(* PLC project Generated.project, CODESYS CODESYS V3.5 SP19 Patch 1 *)
(* stored: creationDateTime 2026-08-11T18:19:14.781842, modificationDateTime 2026-08-11T18:19:14.781842 *)

(* ═══════════════════════════════════════════════════════════════ 🏗️ ST_HardwareImage — Structure globale d'image matérielle (Frontière HwIn) ─────────────────────────────────────────────────────────────── 📄 Lot L5 (Frontière unique HwIn) 🎨 Agrège les 4 sous-domaines matériels : Winch, Translation, Operator, Machine. ═══════════════════════════════════════════════════════════════ *)
TYPE ST_HardwareImage : STRUCT
  Winch : ST_HwWinch;  (* Entrées brutes domaine Treuils M1/M2 + codeurs *)
  Translation : ST_HwTranslation;  (* Entrées brutes domaine Translation M3 + variateur *)
  Operator : ST_HwOperator;  (* Entrées brutes domaine Opérateur / Joystick / bus CAN *)
  Machine : ST_HwMachine;  (* Entrées brutes domaine Sécurités/Communs Machine *)
END_STRUCT;
END_TYPE

(* ═══════════════════════════════════════════════════════════════ 🏗️ ST_HwMachine — Image matérielle brute des entrées communes Machine ─────────────────────────────────────────────────────────────── 📄 Lot L5 (Frontière unique HwIn) 🎨 Regroupe les signaux physiques d'entrée bruts communs à la machine. ═══════════════════════════════════════════════════════════════ *)
TYPE ST_HwMachine : STRUCT
  PowerContactorEngaged_DI : BOOL;  (* Confirm. contacteur puissance engagé *)
  EmergencyChainClosed_DI : BOOL;  (* Boucle AU fermée (coup-de-poing + contact PLC) *)
  PhaseRotationOk_DI : BOOL;  (* Contrôle rotation phases élec. OK *)
  BrakeThermalOk_DI : BOOL;  (* Thermique frein M1/M2/M3 commun OK *)
  M1_M2_KoboldContactFond_DI : BOOL;  (* Retour détecteur fond Kobold *)
  HydraulicThermalOk_DI : BOOL;  (* Thermique centrale hydraulique OK *)
  ConveyorInfeedReady_DI : BOOL;  (* Autorisation démarrage crible (dépôt gravats) *)
END_STRUCT;
END_TYPE

(* ═══════════════════════════════════════════════════════════════ 🏗️ ST_HwOperator — Image matérielle brute des entrées Opérateur / Joystick ─────────────────────────────────────────────────────────────── 📄 Lot L5 (Frontière unique HwIn) 🎨 Regroupe les signaux physiques d'entrée bruts du joystick CANopen JOY1. ═══════════════════════════════════════════════════════════════ *)
TYPE ST_HwOperator : STRUCT
  JoyXRaw_ANA1 : INT;  (* Valeur brute analogique axe X (Translation) *)
  JoyYRaw_ANA2 : INT;  (* Valeur brute analogique axe Y (Levage) *)
  JoyBtnRaw : BOOL;  (* Bouton brut joystick (Homme-Mort) *)
  CanBusState : INT;  (* État bus CANopen (CANbus.GetBusState) *)
  JOY1_DeviceState : DEVICE_STATE;  (* État device JOY1 (GetDeviceState) *)
END_STRUCT;
END_TYPE

(* ═══════════════════════════════════════════════════════════════ 🏗️ ST_HwTranslation — Image matérielle brute des entrées Translation M3 ─────────────────────────────────────────────────────────────── 📄 Lot L5 (Frontière unique HwIn) 🎨 Regroupe les signaux physiques d'entrée bruts de la translation M3 (AC600). ═══════════════════════════════════════════════════════════════ *)
TYPE ST_HwTranslation : STRUCT
  M3_PosTremie_DI : BOOL;  (* Capteur position trémie *)
  M3_PosPV_DI : BOOL;  (* Capteur position point de vitesse (pré-ralentissement) *)
  M3_PosP2_DI : BOOL;  (* Capteur position P2 *)
  M3_PosP1_DI : BOOL;  (* Capteur position P1 *)
  M3_PosMaintenance_DI : BOOL;  (* Capteur position maintenance *)
  M3_BrakeIsOpen_DI : BOOL;  (* Retour frein M3 (1 = ouvert) *)
  M3_ThermalOK_DI : BOOL;  (* 🆕 T96 : retour disjoncteur thermique moteur/variateur AC600 (1 = OK, même polarité que BrakeThermalFeedback/M1/M2ThermalFeedback) — diagnostic seul, l'AC600 se protège déjà lui-même *)
  M3_StatusWord : WORD;  (* Status word variateur AC600 *)
  M3_ActualFrequencyHz : UINT;  (* Fréquence réelle variateur AC600 (x100) *)
  AC600_DeviceState : DEVICE_STATE;  (* État device AC600 (GetDeviceState) *)
END_STRUCT;
END_TYPE

(* ═══════════════════════════════════════════════════════════════ 🏗️ ST_HwWinch — Image matérielle brute des entrées Treuils M1 / M2 ─────────────────────────────────────────────────────────────── 📄 Lot L5 (Frontière unique HwIn) 🎨 Regroupe les signaux physiques d'entrée bruts des treuils M1 et M2. ═══════════════════════════════════════════════════════════════ *)
TYPE ST_HwWinch : STRUCT
  M1_ContactorsReleased_DI : BOOL;  (* Retours contacteurs M1 retombés *)
  M1_ThermalOk_DI : BOOL;  (* Thermique moteur M1 OK *)
  M1_BrakeIsOpen_DI : BOOL;  (* Retour frein M1 (1 = ouvert) *)
  M2_ContactorsReleased_DI : BOOL;  (* Retours contacteurs M2 retombés *)
  M2_ThermalOk_DI : BOOL;  (* Thermique moteur M2 OK *)
  M2_BrakeIsOpen_DI : BOOL;  (* Retour frein M2 (1 = ouvert) *)
  M1M2_TopPositionFree_DI : BOOL;  (* Capteur position haute commun M1/M2 libre *)
  M2_TensionedCable_DI : BOOL;  (* Capteur mou de câble M2 (câble tendu) *)
  COD1_PosValue : UDINT;  (* Valeur brute position codeur COD1 (M1) *)
  COD1_Alarms : UINT;  (* Alarmes brutes COD1 *)
  COD1_Warnings : UINT;  (* Avertissements bruts COD1 *)
  COD1_DeviceState : DEVICE_STATE;  (* État device COD1 (GetDeviceState) *)
  COD2_PosValue : UDINT;  (* Valeur brute position codeur COD2 (M2) *)
  COD2_Alarms : UINT;  (* Alarmes brutes COD2 *)
  COD2_Warnings : UINT;  (* Avertissements bruts COD2 *)
  COD2_DeviceState : DEVICE_STATE;  (* État device COD2 (GetDeviceState) *)
END_STRUCT;
END_TYPE

(* ═══════════════════════════════════════════════════════════════ 🧪 FB_SimBench — Enveloppe unique de simulation pour banc d'essai ─────────────────────────────────────────────────────────────── 📄 Doc métier : DOC/AF/AF_Partie-13_Fonction_Simulation_v2.1.md 📄 Lot L6 (Rebranchement du banc de simulation derrière HwIn) 🎯 Rôle : Compose les 4 blocs de modèle de simulation existants : - FB_Sim_Encoder (instM1, instM2) - FB_Sim_Translation (instTranslation) - FB_Sim_Joystick (instJoystick) - FB_Sim_Safety (instSafety) 🔒 Brique réduite : 0 lecture de variable globale en interne. Toutes les entrées (commandes, stimuli, HwReal) sont passées en paramètres. 🔴 RÈGLES SÉCURITÉ ET POLARITÉ : - Modèle frein M1/M2/M3 : M1_BrakeIsOpen_DI := M1_BrakeCmd (1 = OUVERT). Ne JAMAIS faire NOT BrakeCmd ! (P1 Lot L6). - Retours contacteurs M1/M2 : 1 = tous retombés (TRUE quand RelayFwd=0 et RelayRev=0). ═══════════════════════════════════════════════════════════════ *)
FUNCTION_BLOCK FB_SimBench
  VAR_INPUT
    Enable : BOOL;  (* Activation globale (GVL_Simulation.SimulationModeActive) *)
    M1_RelayFwd : BOOL;  (* ── Commandes issues de l'automate (Scan N-1 / PRG_07 / PRG_10) ────────── *)
    M1_RelayRev : BOOL;
    M1_SpeedContactor_1 : BOOL;  (* 🔧 REX 2026-07-27 : les 4 contacteurs de palier participent au retour unique « tous contacteurs retombés » — sans eux, le modèle annonce l'arrêt alors qu'un palier est encore engagé (fausse condition d'armement Méca A). *)
    M1_SpeedContactor_2 : BOOL;
    M1_SpeedContactor_3 : BOOL;
    M1_SpeedContactor_4 : BOOL;
    M1_SpeedRefPct : REAL;
    M1_PresetTriggerCmd : WORD;
    M1_PresetValueOut : UDINT;
    M1_BrakeCmd : BOOL;  (* TRUE = commande desserrage frein M1 *)
    M2_RelayFwd : BOOL;
    M2_RelayRev : BOOL;
    M2_SpeedContactor_1 : BOOL;  (* 🔧 REX 2026-07-27 : idem M1, voir ci-dessus *)
    M2_SpeedContactor_2 : BOOL;
    M2_SpeedContactor_3 : BOOL;
    M2_SpeedContactor_4 : BOOL;
    M2_SpeedRefPct : REAL;
    M2_PresetTriggerCmd : WORD;
    M2_PresetValueOut : UDINT;
    M2_BrakeCmd : BOOL;  (* TRUE = commande desserrage frein M2 *)
    M3_Direction : INT;  (* 1 = Avant, -1 = Arrière, 0 = Arrêt *)
    M3_SpeedRefPct : REAL;
    M3_BrakeCmd : BOOL;  (* TRUE = commande desserrage frein M3 *)
    M3_TargetNum : INT;  (* Cible sélectionnée (0..4) *)
    PowerKeepAlive_A : BOOL;  (* TRUE = relais A maintenu sagement par le PLC *)
    PowerKeepAlive_B : BOOL;  (* TRUE = relais B maintenu sagement par le PLC *)
    EmergencyArming_RQ : BOOL;  (* Impulsion de réarmement puissance *)
    SimEncoderSpeedFactor : REAL := 1;  (* ── Stimuli & Paramètres de banc ───────────────────────────────────────── *)
    SimSyncDeviationInjectM1 : BOOL := FALSE;
    SimSyncDeviationInjectM2 : BOOL := FALSE;
    SimSyncDeviationOffset_M : REAL := 0.5;
    SimM3SensorsWordActive : BOOL := FALSE;
    SimM3SensorsWord : BYTE := 16#01;
    SimJoystickRawX : INT := 5000;
    SimJoystickRawY : INT := 5000;
    SimJoystickRawButton : BOOL := FALSE;
    SimKoboldContactValue : BOOL := FALSE;
    BtnEmergencyStop : BOOL := FALSE;  (* Simulation appui coup-de-poing AU *)
    HwReal : ST_HardwareImage;  (* ── Image réelle fallback ──────────────────────────────────────────────── *)
  END_VAR
  VAR_OUTPUT
    Winch : ST_HwWinch;
    Translation : ST_HwTranslation;
    Operator : ST_HwOperator;
    Machine : ST_HwMachine;
  END_VAR
  VAR_IN_OUT
    RawPosM1 : UDINT;  (* Mémoire _SimEncoderRawPosM1 dans GVL_PERSISTENT *)
    RawPosM2 : UDINT;  (* Mémoire _SimEncoderRawPosM2 dans GVL_PERSISTENT *)
  END_VAR
  VAR
    instSimEncoderM1 : FB_Sim_Encoder;  (* Modèles sous-jacents *)
    instSimEncoderM2 : FB_Sim_Encoder;
    instSimTranslation : FB_Sim_Translation;
    instSimJoystick : FB_Sim_Joystick;
    instSimSafety : FB_Sim_Safety;
    M1_PresetCmd : BOOL;  (* Calculs internes *)
    M2_PresetCmd : BOOL;
    M1_OffsetPts : DINT;
    M2_OffsetPts : DINT;
    M3_RelayFwd : BOOL;
    M3_RelayRev : BOOL;
    M3_ActualFreqHz : UINT;
    M3_StatusWordSim : WORD;
  END_VAR

            

// === IMPLEMENTATION ===

IF NOT Enable THEN
    Winch       := HwReal.Winch;
    Translation := HwReal.Translation;
    Operator    := HwReal.Operator;
    Machine     := HwReal.Machine;
    RETURN;
END_IF;


// ── 1. MODÈLE TREUILS (M1 + M2) ─────────────────────────────────────────────
// Presets codeurs : déclenchés si PresetTriggerCmd = 2
M1_PresetCmd := (M1_PresetTriggerCmd = 2);
M2_PresetCmd := (M2_PresetTriggerCmd = 2);

// Conversions d'injection d'écart synchro (0.5m -> points codeur avec 8192 pts/tour, 2m/tour)
// 1m = 4096 points codeur.
M1_OffsetPts := REAL_TO_DINT(SimSyncDeviationOffset_M * 4096.0);
M2_OffsetPts := REAL_TO_DINT(SimSyncDeviationOffset_M * 4096.0);

// Instance modèle codeur M1
instSimEncoderM1(
    Enable           := TRUE,
    RelayFwd         := M1_RelayFwd,
    RelayRev         := M1_RelayRev,
    SpeedRefPct      := M1_SpeedRefPct,
    PresetCmd        := M1_PresetCmd,
    PresetValue      := M1_PresetValueOut,
    SpeedScaleFactor := SimEncoderSpeedFactor,
    TestOffsetCmd    := SimSyncDeviationInjectM1,
    TestOffsetPts    := M1_OffsetPts,
    RawPos           := RawPosM1
);

// Instance modèle codeur M2
instSimEncoderM2(
    Enable           := TRUE,
    RelayFwd         := M2_RelayFwd,
    RelayRev         := M2_RelayRev,
    SpeedRefPct      := M2_SpeedRefPct,
    PresetCmd        := M2_PresetCmd,
    PresetValue      := M2_PresetValueOut,
    SpeedScaleFactor := SimEncoderSpeedFactor,
    TestOffsetCmd    := SimSyncDeviationInjectM2,
    TestOffsetPts    := M2_OffsetPts,
    RawPos           := RawPosM2
);

// Recopie structures Winch simulées :
// 🛑 POLARITÉ DE FREIN SIMULÉ (P1 Lot L6) : 1 = contacteur commandé = frein OUVERT.
// Câblage réel : DI = 1 ⟺ frein OUVERT. Le modèle produit donc M1_BrakeIsOpen_DI := M1_BrakeCmd !
Winch.M1_BrakeIsOpen_DI        := M1_BrakeCmd;
// 🔧 REX 2026-07-27 : retour UNIQUE « tous contacteurs retombés » = sens ET vitesse.
// Omettre les paliers ferait croire à l'arrêt pendant les transitoires → Méca A armée à tort.
Winch.M1_ContactorsReleased_DI := NOT (M1_RelayFwd OR M1_RelayRev
                                    OR M1_SpeedContactor_1 OR M1_SpeedContactor_2
                                    OR M1_SpeedContactor_3 OR M1_SpeedContactor_4);
Winch.M1_ThermalOk_DI          := TRUE; // Sauf panne simulée

Winch.M2_BrakeIsOpen_DI        := M2_BrakeCmd;
Winch.M2_ContactorsReleased_DI := NOT (M2_RelayFwd OR M2_RelayRev
                                    OR M2_SpeedContactor_1 OR M2_SpeedContactor_2
                                    OR M2_SpeedContactor_3 OR M2_SpeedContactor_4);
Winch.M2_ThermalOk_DI          := TRUE;

Winch.M1M2_TopPositionFree_DI  := TRUE; // Butée libre au repos en simu
Winch.M2_TensionedCable_DI     := TRUE; // Câble tendu en simu

Winch.COD1_PosValue            := instSimEncoderM1.RawPosOut;
Winch.COD1_Alarms              := 0;
Winch.COD1_Warnings            := 0;
Winch.COD1_DeviceState         := 4; // DEVICE_STATE RUNNING = 4 (bus OK)

Winch.COD2_PosValue            := instSimEncoderM2.RawPosOut;
Winch.COD2_Alarms              := 0;
Winch.COD2_Warnings            := 0;
Winch.COD2_DeviceState         := 4; // DEVICE_STATE RUNNING = 4


// ── 2. MODÈLE TRANSLATION M3 (AC600) ─────────────────────────────────────────
M3_RelayFwd := (M3_Direction = 1);
M3_RelayRev := (M3_Direction = -1);

instSimTranslation(
    Enable      := TRUE,
    TargetNum   := M3_TargetNum,
    RelayFwd    := M3_RelayFwd,
    RelayRev    := M3_RelayRev,
    TravelTimeS := 8.0,
    PVLeadTimeS := 2.0
);

// Remplissage capteurs de position M3 :
IF SimM3SensorsWordActive THEN
    Translation.M3_PosTremie_DI      := SimM3SensorsWord.0;
    Translation.M3_PosPV_DI          := SimM3SensorsWord.1;
    Translation.M3_PosP2_DI          := SimM3SensorsWord.2;
    Translation.M3_PosP1_DI          := SimM3SensorsWord.3;
    Translation.M3_PosMaintenance_DI := SimM3SensorsWord.4;
ELSE
    Translation.M3_PosTremie_DI      := instSimTranslation.PosTremie;
    Translation.M3_PosPV_DI          := instSimTranslation.PosPV;
    Translation.M3_PosP2_DI          := instSimTranslation.PosP2;
    Translation.M3_PosP1_DI          := instSimTranslation.PosP1;
    Translation.M3_PosMaintenance_DI := instSimTranslation.PosMaintenance;
END_IF;

// Polarité frein M3 (1 = OUVERT)
Translation.M3_BrakeIsOpen_DI    := M3_BrakeCmd;

// 🆕 T96 : thermique moteur/variateur AC600 — pas de panne simulée, toujours OK (comme Winch.M1/M2_ThermalOk_DI)
Translation.M3_ThermalOK_DI      := TRUE;

// Simulation StatusWord AC600 : Bit 0 (Power Ready) = 1, Bit 7 (Comm Ready) = 1 -> 16#0081
IF (M3_Direction <> 0) THEN
    M3_StatusWordSim := 16#0087; // + Operating/Running
    M3_ActualFreqHz  := REAL_TO_UINT(M3_SpeedRefPct * 50.0); // 50.0 Hz à 100% (x100 -> 5000)
ELSE
    M3_StatusWordSim := 16#0081;
    M3_ActualFreqHz  := 0;
END_IF;

Translation.M3_StatusWord        := M3_StatusWordSim;
Translation.M3_ActualFrequencyHz := M3_ActualFreqHz;
Translation.AC600_DeviceState    := 4; // DEVICE_STATE RUNNING = 4


// ── 3. MODÈLE OPÉRATEUR / JOYSTICK ───────────────────────────────────────────
instSimJoystick(
    Enable     := TRUE,
    NeutralRaw := 5000,
    MaxRaw     := 10000
);

// Permet aux stimuli de banc de surcharger le retour du joystick si spécifié :
IF SimJoystickRawX <> 5000 THEN
    Operator.JoyXRaw_ANA1 := SimJoystickRawX;
ELSE
    Operator.JoyXRaw_ANA1 := instSimJoystick.RawX;
END_IF;

IF SimJoystickRawY <> 5000 THEN
    Operator.JoyYRaw_ANA2 := SimJoystickRawY;
ELSE
    Operator.JoyYRaw_ANA2 := instSimJoystick.RawY;
END_IF;

IF SimJoystickRawButton THEN
    Operator.JoyBtnRaw := TRUE;
ELSE
    Operator.JoyBtnRaw := instSimJoystick.RawButton;
END_IF;

Operator.CanBusState      := 2; // CANbusState 2 = ACTIVE (confirmé terrain)
Operator.JOY1_DeviceState := 4; // DEVICE_STATE RUNNING = 4


// ── 4. MODÈLE SÉCURITÉ & COMMUNS MACHINE ─────────────────────────────────────
instSimSafety(
    Enable           := TRUE,
    PowerCutOff_A    := PowerKeepAlive_A,
    PowerCutOff_B    := PowerKeepAlive_B,
    EmergencyArming  := EmergencyArming_RQ,
    BtnEmergencyStop := BtnEmergencyStop
);

Machine.PowerContactorEngaged_DI   := instSimSafety.SimContactorOk;
Machine.EmergencyChainClosed_DI    := instSimSafety.SimChainOk;
Machine.PhaseRotationOk_DI         := TRUE;
Machine.BrakeThermalOk_DI          := TRUE;
Machine.M1_M2_KoboldContactFond_DI := SimKoboldContactValue;
Machine.HydraulicThermalOk_DI      := TRUE;

          
END_FUNCTION_BLOCK

(* ═══════════════════════════════════════════════════════════════ 🧪 FB_Sim_Encoder — Simulation physique d'un codeur absolu de treuil ─────────────────────────────────────────────────────────────── 📄 Doc métier : DOC/AF/AF_Partie-13_Fonction_Simulation_v2.1.md 🧩 Brique réduite (Partie3 §1bis, "briques E/S & diagnostics") : pas de contrat Enable/Reset/Error complet, pas de StartStop/SafeStop — outil de banc, pas du métier machine. 🎯 Rôle : fait "compter" un codeur absolu comme si le treuil tournait réellement, à partir des relais de sens commandés et de la vitesse rampée courante. Extraction PURE de la logique déjà en place dans `PRG_02_Encoders.st` (bloc "SIMULATION SUR BANC DE TEST") — aucun changement de comportement, juste la dissociation en FB dédié. 📥 Enable : simulation active (SimulationModeActive AND NOT BusEncoderMxIsReal) 📥 RelayFwd/RelayRev : sens commandé (contacteurs de sens du treuil) 📥 SpeedRefPct : vitesse rampée courante (magnitude, %) — ex. instWinchM1.SpeedRamp.Current 📥 PresetCmd : TRUE le cycle où un preset (homing) doit être appliqué (PresettTrigCmd = 2) 📥 PresetValue : valeur brute à charger lors du preset 📥 SpeedScaleFactor : 🔧 REX 2026-07-07 — multiplicateur de vitesse simulation (confort de test banc uniquement, sans rapport avec une calibration réelle). Défaut 1.0 = comportement d'origine. Câblé sur GVL_Simulation.TstEncoderSpeedFactor (réglable à chaud, sans recompiler). 📤 RawPosOut : position brute simulée (UDINT), à aiguiller à la place de la valeur EtherCAT réelle quand le device n'est pas Operational (voir PRG_02_Encoders.st) 🔧 REX 2026-07-08 : `RawPos` déplacé en `VAR_IN_OUT`, référencé depuis `GVL_PERSISTENT` (même pattern que `Calib` dans `FB_Encoder_Homing`) — `PERSISTENT` n'est valide que sur du `VAR_GLOBAL` en CODESYS, pas sur une variable locale de FB (tenté en `VAR RETAIN` puis `VAR PERSISTENT RETAIN` locaux, aucun des deux ne convient). Un vrai codeur absolu physique conserve son comptage brut même à travers un reset FROID (indépendant de l'automate) — il fallait donc bien du PERSISTENT RETAIN réel, regroupé avec le reste dans GVL_PERSISTENT. ═══════════════════════════════════════════════════════════════ === DECLARATION (à coller dans la partie déclaration du POU FB_Sim_Encoder) === *)
FUNCTION_BLOCK FB_Sim_Encoder
  VAR_INPUT
    Enable : BOOL;
    RelayFwd : BOOL;
    RelayRev : BOOL;
    SpeedRefPct : REAL;
    PresetCmd : BOOL;
    PresetValue : UDINT;
    SpeedScaleFactor : REAL := 1;  (* 🔧 REX 2026-07-07 — confort de test, voir bandeau ci-dessus *)
    TestOffsetCmd : BOOL;  (* 🆕 REX 2026-07-08 (4) — front montant = applique TestOffsetPts (test banc) *)
    TestOffsetPts : DINT := 0;  (* 🆕 REX 2026-07-08 (4) — décalage signé à appliquer (points bruts) *)
  END_VAR
  VAR_OUTPUT
    RawPosOut : UDINT;
  END_VAR
  VAR_IN_OUT
    RawPos : UDINT;  (* 🔧 REX 2026-07-08 : référence _SimEncoderRawPosM1/M2 (survit au reset froid) *)
  END_VAR
  VAR
    Increment : UDINT;  (* 🔧 REX 2026-07-07 — évite de dupliquer le calcul 2x *)
    TestOffsetEdge : R_TRIG;  (* 🆕 REX 2026-07-08 (4) *)
  END_VAR

            

// === IMPLEMENTATION (à coller dans le corps ST du POU FB_Sim_Encoder) ===

IF NOT Enable THEN
    RawPosOut := RawPos;
    RETURN;
END_IF;

// 🆕 REX 2026-07-08 (4) — injection test banc : VRAI saut de position (comme un glissement réel),
// pour tester Concept 1 / Méca E ET le rattrapage joystick (voir GVL_Simulation bandeau).
TestOffsetEdge(CLK := TestOffsetCmd);
IF TestOffsetEdge.Q THEN
    RawPos := DINT_TO_UDINT(UDINT_TO_DINT(RawPos) + TestOffsetPts);
END_IF;

Increment := REAL_TO_UDINT(SpeedRefPct * 0.1 * SpeedScaleFactor);

IF PresetCmd THEN
    RawPos := PresetValue;
ELSIF RelayFwd THEN
    RawPos := RawPos + Increment;
ELSIF RelayRev THEN
    IF RawPos >= Increment THEN
        RawPos := RawPos - Increment;
    ELSE
        RawPos := 0;
    END_IF;
END_IF;

RawPosOut := RawPos;

          
END_FUNCTION_BLOCK

(* ═══════════════════════════════════════════════════════════════ 🧪 FB_Sim_Joystick — Simulation des entrées brutes joystick (bus CAN hors ligne) ─────────────────────────────────────────────────────────────── 📄 Doc métier : DOC/AF/AF_Partie-13_Fonction_Simulation_v2.1.md 🧩 Brique réduite (Partie3 §1bis) : outil de banc, pas du métier machine. 🎯 Rôle : remplace l'ancien bypass homme-mort codé en dur dans `FB_Joystick` (`GVL_DEBUG.DBG_DeadmanBypass_TEST`, qui forçait `DeadmanArmed` en permanence — un vrai contournement de sécurité). Ici, on simule les ENTRÉES BRUTES du capteur (`RawX`/`RawY`/`RawButton`) : le homme-mort réel de `FB_Joystick` reste pleinement actif et doit toujours être "actionné" (forcer `RawButton` en instance CODESYS) pour armer — comportement métier testé pour de vrai, pas contourné. 📥 Enable : simulation active (SimulationModeActive AND NOT BusJoystickSignalIsReal) — 🔧 REX 2026-07-08 : granularité séparée du bus CANopen (BusJoystickIsReal, voir GVL_Simulation) 📥 NeutralRaw : valeur brute simulée au repos (voir GVL_Simulation.TstJoystickForceNeutralRaw) 📥 MaxRaw : valeur brute simulée à fond (voir GVL_Simulation.TstJoystickForceMaxRaw) 📤 RawX/RawY : forçables en instance CODESYS (par défaut = NeutralRaw, repos) 📤 RawButton : forçable en instance CODESYS (par défaut = FALSE, relâché) 💡 Note d'application : en vue instance CODESYS, forcer `RawX`/`RawY` à `MaxRaw` (ou une valeur intermédiaire) pour simuler un débattement, et `RawButton` à `TRUE` pour simuler l'appui homme-mort — exactement comme on forcerait le vrai capteur. ═══════════════════════════════════════════════════════════════ === DECLARATION (à coller dans la partie déclaration du POU FB_Sim_Joystick) === *)
FUNCTION_BLOCK FB_Sim_Joystick
  VAR_INPUT
    Enable : BOOL;
    NeutralRaw : INT := 5000;
    MaxRaw : INT := 10000;
  END_VAR
  VAR_OUTPUT
    RawX : INT;  (* 🔧 Forçable en instance CODESYS (repos = NeutralRaw) *)
    RawY : INT;  (* 🔧 Forçable en instance CODESYS (repos = NeutralRaw) *)
    RawButton : BOOL;  (* 🔧 Forçable en instance CODESYS (repos = FALSE) *)
  END_VAR
  VAR
    FirstCycle : BOOL := TRUE;
  END_VAR

            

// === IMPLEMENTATION (à coller dans le corps ST du POU FB_Sim_Joystick) ===

// 🔑 Initialise au neutre au premier cycle uniquement — ensuite RawX/RawY/RawButton
// restent forçables librement en instance CODESYS (un Force n'est jamais écrasé par TRUE,
// mais une simple écriture cyclique l'écraserait — donc pas de ré-assignation continue ici).
IF NOT Enable THEN
    FirstCycle := TRUE;
    RETURN;
END_IF;

IF FirstCycle THEN
    RawX := NeutralRaw;
    RawY := NeutralRaw;
    RawButton := FALSE;
    FirstCycle := FALSE;
END_IF;

          
END_FUNCTION_BLOCK

(* ═══════════════════════════════════════════════════════════════ 🧪 FB_Sim_Safety — Simulation de la chaîne d'AU et du contacteur de puissance ─────────────────────────────────────────────────────────────── 📥 Enable : activation de la simulation (SimulationModeActive AND NOT SensorEmergencyStopChainIsReal) 📥 PowerCutOff_A : demande de coupure PLC canal A (maintenu à TRUE en marche normale) 📥 PowerCutOff_B : demande de coupure PLC canal B (maintenu à TRUE en marche normale) 📥 EmergencyArming : impulsion de réarmement (EmergencyArming_RQ) 📤 SimChainOk : simulation de la boucle AU (boutons relâchés et coupures PLC inactives) 📤 SimContactorOk : simulation du contacteur engagé (PowerContactorEngaged) ⚙️ Logique physique : - La chaîne d'AU (SimChainOk) est saine si les deux relais PLC de coupure sont maintenus fermés (TRUE). - Le contacteur s'engage (SimContactorOk) lors d'une impulsion de réarmement (EmergencyArming) et s'auto-maintient tant que la chaîne reste saine (SimChainOk). - Toute coupure de la chaîne (SimChainOk = FALSE) fait retomber immédiatement le contacteur. ═══════════════════════════════════════════════════════════════ 📄 Docs : DOC/AF/AF_Partie-13_Fonction_Simulation_v2.1.md *)
FUNCTION_BLOCK FB_Sim_Safety
  VAR_INPUT
    Enable : BOOL;  (* Activation de la simulation *)
    PowerCutOff_A : BOOL;  (* Commande coupure canal A (TRUE = OK/fermé) *)
    PowerCutOff_B : BOOL;  (* Commande coupure canal B (TRUE = OK/fermé) *)
    EmergencyArming : BOOL;  (* Impulsion de réarmement (TRUE = pulse) *)
    BtnEmergencyStop : BOOL;  (* Force l'ouverture de la boucle (TRUE = bouton appuyé/défaut) *)
  END_VAR
  VAR_OUTPUT
    SimChainOk : BOOL;  (* Boucle AU simulée saine *)
    SimContactorOk : BOOL;  (* Contacteur simulé engagé *)
  END_VAR
  VAR
    ContactorLatch : BOOL;  (* Mémorisation de l'auto-maintien du contacteur *)
  END_VAR

            

// === IMPLEMENTATION ===
IF NOT Enable THEN
    SimChainOk     := FALSE;
    SimContactorOk := FALSE;
    ContactorLatch := FALSE;
    RETURN;
END_IF;

// 1. La chaîne AU est saine si le PLC maintient les deux relais de coupure de puissance
// AND if no emergency stop button is pressed (BtnEmergencyStop is FALSE)
SimChainOk := PowerCutOff_A AND PowerCutOff_B AND NOT BtnEmergencyStop;

// 2. Logique d'auto-maintien (latch) du contacteur avec priorité à la coupure
IF NOT SimChainOk THEN
    ContactorLatch := FALSE;
ELSIF EmergencyArming THEN
    ContactorLatch := TRUE;
END_IF;

// Recopie vers la sortie
SimContactorOk := ContactorLatch;

          
END_FUNCTION_BLOCK

(* ═══════════════════════════════════════════════════════════════ 🧪 FB_Sim_Translation — Simulation dynamique du trajet translation M3 (temps de parcours) ─────────────────────────────────────────────────────────────── 📄 Doc métier : DOC/AF/AF_Partie-13_Fonction_Simulation_v2.1.md 🧩 Brique réduite (Partie3 §1bis) : outil de banc, pas du métier machine. 🎯 Rôle : remplace le forçage manuel du capteur de position cible en vue instance CODESYS (voir `GVL_Translation_M3_Stub.st`, doc Partie11 §9bis) par une simulation par temps de parcours : le translation "arrive" à la cible sélectionnée (`TargetNum`) après `TravelTimeS` secondes de commande continue dans le bon sens (`RelayFwd`/`RelayRev`). Non prioritaire (M3 translation) — treuils/benne/codeurs sont la priorité de ce lot. 📥 Enable : simulation active (SimulationModeActive AND NOT SensorTranslationPositionIsReal) 📥 TargetNum : cible sélectionnée (0=Aucun, 1=Trémie, 2=P2, 3=P1, 4=Maintenance) — réutilise `GVL_Translation_M3_Stub.StubTranslationPositionSelect_IHM` — 🆕 REX 2026-07-18 : PV n'est JAMAIS une cible sélectionnable (point de ralentissement uniquement, pas d'arrêt), voir AF_Partie-02 v2.12 §3bis 📥 RelayFwd/RelayRev : sens déduit du mot de commande EtherCAT M3 📥 TravelTimeS : temps de trajet simulé (s) — défaut 8.0 (fourchette 5-10s validée utilisateur, pas de donnée réelle pour calibrer plus précisément) 📥 PVLeadTimeS : durée (s) avant la fin du trajet Trémie où PV s'active (approche) 📤 PosTremie/PosPV/PosP2/PosP1/PosMaintenance : TRUE quand la cible (ou le point de ralentissement PV) correspondante est atteinte — à OR'er sur le `InputRaw` du capteur réel correspondant (`PRG_02_Acquisition.HwIn`). ⏱️ Changement de cible (`TargetNum`) → trajet remis à zéro (redémarre du début). Relais retombés (ni Fwd ni Rev) → progression mise EN PAUSE (pas remise à zéro). ═══════════════════════════════════════════════════════════════ === DECLARATION (à coller dans la partie déclaration du POU FB_Sim_Translation) === *)
FUNCTION_BLOCK FB_Sim_Translation
  VAR_INPUT
    Enable : BOOL;
    TargetNum : INT;
    RelayFwd : BOOL;
    RelayRev : BOOL;
    TravelTimeS : REAL := 8;
    PVLeadTimeS : REAL := 2;
  END_VAR
  VAR_OUTPUT
    PosTremie : BOOL;
    PosPV : BOOL;
    PosP2 : BOOL;
    PosP1 : BOOL;
    PosMaintenance : BOOL;
  END_VAR
  VAR
    CycleTimeCalc : FB_CycleTime;  (* 📚 Réutilisation — pas de recalcul maison du temps de cycle *)
    ElapsedS : REAL;
    LastTargetNum : INT;
    TargetChanged : BOOL;
    Reached : BOOL;
  END_VAR

            

// === IMPLEMENTATION (à coller dans le corps ST du POU FB_Sim_Translation) ===

IF NOT Enable THEN
    ElapsedS := 0.0;
    LastTargetNum := TargetNum;
    PosTremie := FALSE; PosPV := FALSE; PosP2 := FALSE; PosP1 := FALSE; PosMaintenance := FALSE;
    RETURN;
END_IF;

CycleTimeCalc(DefaultValueS := 0.010);

// 🔁 Changement de cible = nouveau trajet, on repart de zéro
TargetChanged := (TargetNum <> LastTargetNum);
LastTargetNum := TargetNum;
IF TargetChanged THEN
    ElapsedS := 0.0;
END_IF;

// ⏱️ Progression du trajet UNIQUEMENT si un relais de sens est actif (mouvement réel demandé) ;
// à l'arrêt, la progression reste EN PAUSE (pas remise à zéro).
IF (RelayFwd OR RelayRev) AND (ElapsedS < TravelTimeS) THEN
    ElapsedS := ElapsedS + CycleTimeCalc.CycleTimeS;
    IF ElapsedS > TravelTimeS THEN
        ElapsedS := TravelTimeS;
    END_IF;
END_IF;

Reached := (ElapsedS >= TravelTimeS);

// 🆕 REX 2026-07-18 : les capteurs sont codés par progression monotone.
// La simulation doit donc produire un mot valide à chaque instant, et non
// uniquement activer le capteur de la cible. Le mot est :
//   11111 Trémie | 01111 PV | 00111 P2 | 00011 P1 | 00001 approche Maintenance | 00000 Maintenance.
// 🔧 REX 2026-07-21 : au repos / boot (TargetNum = 0), la position neutre par défaut
// est positionnée sur P2 (00111) pour éviter d'être par défaut sur le fin de course extrême Maintenance (00000).
PosTremie := FALSE;
PosPV := FALSE;

IF TargetNum = 0 THEN
    // Position neutre par défaut au boot (P2 = 00111) — évite le fin de course extrême arrière au démarrage
    PosP2 := TRUE;
    PosP1 := TRUE;
    PosMaintenance := TRUE;
ELSIF TargetNum = 1 THEN
    // Trajet vers Trémie : PV puis Trémie, avec les trois capteurs de droite actifs.
    PosP2 := FALSE; PosP1 := FALSE; PosMaintenance := FALSE;
    IF ElapsedS >= (TravelTimeS - PVLeadTimeS) THEN
        PosPV := TRUE;
        PosP2 := TRUE;
        PosP1 := TRUE;
        PosMaintenance := TRUE;
    END_IF;
    IF Reached THEN
        PosTremie := TRUE;
    END_IF;
ELSIF TargetNum = 2 THEN
    // P2 = 00111
    PosP2 := TRUE;
    PosP1 := TRUE;
    PosMaintenance := TRUE;
ELSIF TargetNum = 3 THEN
    // P1 = 00011
    PosP2 := FALSE;
    PosP1 := TRUE;
    PosMaintenance := TRUE;
ELSIF TargetNum = 4 THEN
    // Maintenance = 00000 : PosMaintenance reste FALSE pour respecter le codage.
    PosP2 := FALSE;
    PosP1 := FALSE;
    PosMaintenance := FALSE;
ELSE
    PosP2 := TRUE;
    PosP1 := TRUE;
    PosMaintenance := TRUE;
END_IF;

          
END_FUNCTION_BLOCK

(* ═══════════════════════════════════════════════════════════════ ⏱️ FB_CycleTime — Mesure du temps de cycle réel de la tâche ─────────────────────────────────────────────────────────────── 📄 Doc métier : DOC/AF/AF_Partie-08_Fonction_Joystick_v2.0.md §2 (base de temps utilisée par FB_Filter_PT1, composé dans FB_Joystick) ═══════════════════════════════════════════════════════════════ *)
FUNCTION_BLOCK FB_CycleTime
  VAR_INPUT
    DefaultValueS : REAL := 0.004;  (* Valeur de secours par défaut (ex. 4ms) *)
  END_VAR
  VAR_OUTPUT
    CycleTimeS : REAL;  (* Temps écoulé réel calculé (secondes) *)
  END_VAR
  VAR
    TimeCurrent : TIME;  (* Temps système actuel *)
    TimeLast : TIME;  (* Empreinte de temps du cycle précédent *)
    DeltaTimeMs : UDINT;  (* Écart brut calculé (ms) *)
    InitDone : BOOL;  (* Drapeau d'initialisation du premier cycle *)
  END_VAR

            

// 1. ACQUISITION DU TEMPS SYSTÈME
TimeCurrent := TIME();

// 2. INITIALISATION UNIQUE AU PREMIER CYCLE
IF NOT InitDone THEN
    TimeLast := TimeCurrent;
    InitDone := TRUE;
    CycleTimeS := DefaultValueS;
    RETURN;
END_IF;

// 3. CALCUL DU DELTA EN MILLISECONDES
DeltaTimeMs := TIME_TO_UDINT(TimeCurrent - TimeLast);

// 4. CONVERSION ET CHARGE DE SECOURS
IF DeltaTimeMs > 0 THEN
    CycleTimeS := UDINT_TO_REAL(DeltaTimeMs) / 1000.0;
ELSE
    CycleTimeS := DefaultValueS;
END_IF;

// 5. ARCHIVAGE POUR LE PROCHAIN CYCLE
TimeLast := TimeCurrent;

          
END_FUNCTION_BLOCK
